{attribute addProperty BoxType "AT2050-5500-0018"}
{attribute addProperty Id "ControlAT %Q*UINT162"}
{attribute addProperty CRC "1934178468"}
{attribute addProperty SizeInBites "16"}
{attribute addProperty SizeInBytes "2"}
TYPE FB_Outputs_734938A4 :
STRUCT
	{attribute addProperty Name "Control"}
	Control AT %Q* : UINT;
END_STRUCT
END_TYPE

(* stored: Version 1.2.0.0, ProductVersion 3.1.4024.9
   DUT FB_Outputs_734938A4: Id {81474b37-a7f8-4432-8c83-1a04cf4b891e} *)
